FUNCTION_BLOCK FB_Blinking
VAR_INPUT
END_VAR
VAR_OUTPUT	
	
END_VAR
VAR
	ton1		:TON;
END_VAR

METHOD M_Blink : BOOL
VAR_OUTPUT
	bBlink		:BOOL;
END_VAR
ton1(IN:= NOT ton1.Q, PT:= T#1S, Q=> , ET=> );

IF	ton1.Q THEN
	ton1(IN:= FALSE, PT:= T#1S, Q=> , ET=> );	
	bBlink := NOT bBlink;
END_IF
END_METHOD

END_FUNCTION_BLOCK

(* stored: Version 1.1.0.1, ProductVersion 3.1.4022.16
   POU FB_Blinking: Id {3473e3f0-5203-43a5-b6b5-63c2e9220496}, SpecialFunc None
   Method M_Blink: Id {ebc06794-fd21-4ea2-8b38-b16fe10121ec} *)
